FUNCTION "sndCALIBR&Tara" : Void
{ S7_Optimized_Access := 'TRUE' }
VERSION : 0.1
   VAR_INPUT
      ADDR_DEVICE : UInt;   // адрес опрашиваемого устройства
      ton_changeStep : Bool;   // таймер на переход следующего шага опроса
   END_VAR

   VAR_IN_OUT
      MB_MASTER : Struct
         REQ : Bool;
         MB_ADDR : UInt;
         MODE : USInt;
         DATA_ADDR : UDInt;
         DATA_LEN : UInt;
         DONE : Bool;
         BUSY : Bool;
         ERROR : Bool;
      END_STRUCT;
      Ton_Start : Bool;   // сигнал на старт таймера
      Buffer : Array[0..20] of Word;   // буффер данных у блока мастера модбаса
      Step : SInt;   // текущий шаг
      Calibrate : Bool;   // сигнал на калибровку
      Tara : Bool;   // сигнал на тарирование
   END_VAR


BEGIN
	        IF #Calibrate OR//калибровка
	            #Tara//тарирование
	        THEN
	            #Ton_Start := TRUE;

	            #MB_MASTER.MB_ADDR := #ADDR_DEVICE;
	            #MB_MASTER.MODE := 1;
	            #MB_MASTER.DATA_ADDR := 40068;
	            #MB_MASTER.DATA_LEN := 1;
	            #MB_MASTER.REQ := TRUE;

	            IF #Calibrate THEN
	                #Buffer[0] := 16#C2FA;
	            ELSIF #Tara THEN
	                #Buffer[0] := 16#C1BA;
	            END_IF;

	            IF NOT (#MB_MASTER.BUSY) AND
	                (#MB_MASTER.DONE OR
	                #ton_changeStep OR
	                #MB_MASTER.ERROR) THEN
	                #MB_MASTER.REQ := FALSE;
	                #Ton_Start := FALSE;
	                #Step := #Step + 1;
	                IF #Calibrate THEN
	                    #Calibrate := FALSE;
	                ELSIF #Tara THEN
	                    #Tara := false;
	                END_IF;

	                #Buffer[0] := 0;
	            END_IF;
	        ELSE
	            #Step := #Step + 1;
	            #MB_MASTER.REQ := FALSE;
	        END_IF;



END_FUNCTION

